Staubli VAL3: uInitTRSF.pgx

program uInitTRSF(trsf& x_TRSF[] (dimensions=1))
begin
  x_TRSF[0]=swap:trWinUp[0]
  x_TRSF[1]=swap:trWinUp[1]
  x_TRSF[2]=swap:trWinDown[0]
  x_TRSF[3]=swap:trWinDown[1]
end
